FUNCTION_BLOCK EQ_BOOL (* IEC 61131-3 BOOL equality test *)
  (* Standard: 61131-3 *)
  (* Version 0.0, 2006-09-14, JHC, Holobloc Inc *)
  (* Compiler header: package fb.rt.plc.bits; *)
  (* Compiler classdef: (i1 == i2) *)
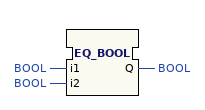
  VAR_INPUT
    i1 : BOOL;
    i2 : BOOL;
  END_VAR
  VAR_OUTPUT
    Q : BOOL;
  END_VAR
END_FUNCTION_BLOCK
